{attribute 'qualified_only'}
{attribute 'strict'}
{attribute 'to_string'}
TYPE EN_TapeInSystemStatus :
(
	tapeOnlyInPickPlate,
	tapeGrippedInPicker,
	tapeCutted,
	tapeOnApplyPlates
);
END_TYPE

(* stored: Version 1.1.0.1, ProductVersion 3.1.4024.12
   DUT EN_TapeInSystemStatus: Id {026e0f87-f8b7-41ac-bd0e-ccfbc49978ca} *)
